PROGRAM MAIN
VAR

	xResetCounters				:BOOL;
	LocalEcDevState		AT%I*	:UINT ;
	EncoderLoopBack				:ARRAY[1..NumOfEcMasters] OF FB_EncoderLoopBack;
END_VAR

VAR_TEMP
	i						:UDINT;
END_VAR

PRG_EcDiag();

FOR i:=1 TO NumOfEcMasters DO
	EncoderLoopBack[i]();
END_FOR

IF xResetCounters THEN
	xResetCounters:=FALSE;
	FOR i:=1 TO NumOfEcMasters DO
		EncoderLoopBack[i].Reset();
	END_FOR
END_IF

END_PROGRAM

(* stored: Version 1.1.0.1, ProductVersion 3.1.4024.11
   POU MAIN: Id {c53a4bec-71d5-4e96-ba06-f49f987385ba}, SpecialFunc None *)
